// TIA Portal V20 export
FUNCTION_BLOCK "FB_Send_Water_Fountain_To_Rework"   // FB7, LAD
{ S7_Optimized_Access := 'TRUE' }
// stored: AutoNumber false, MemoryReserve 100, SetENOAutomatically false
   VAR_INPUT
      Emergency_Stop_Release : Bool;
      Start : Bool;
      Water_Fountain_Fail_Test : Bool;
      Trigger_Read_Serial_Number_Exit_Functional_Test : Bool;
      Sensor_Water_Fountain_Exit_Functional_Test_Spinner_Conveyor_Belt : Bool;
      Sensor_Spinner_Exit_Functional_Test_Position_Withdrawn : Bool;
      Sensor_Spinner_Exit_Functional_Test_Position_Advanced : Bool;
      Sensor_Water_Fountain_Exit_Functional_Test_After_Spinner_Conveyor_Belt : Bool;
      Sensor_Water_Fountain_Geting_Entrace_Rework_Conveyor_Belt_Start : Bool;
   END_VAR
   VAR_OUTPUT
      Turn_On_Conveyor_Belt_Motor_Spinner_Get_Exit_Functional_Test : Bool;
      Valve_Advance_Spinner_Get_Exit_Functional_Test : Bool;
      Pause_Conveyor_Belt_And_Carousel_Functional_Test : Bool;
   END_VAR
   VAR
      Aux_Trig_0 : Bool;
      Aux_Trig_1 : Bool;
      Aux_Trig_2 : Bool;
      Aux_Trig_3 : Bool;
      Aux_Trig_4 : Bool;
      Aux_Trig_5 : Bool;
      Aux_Trig_6 : Bool;
      Aux_Trig_7 : Bool;
      Wait_Clean_Spinner : Bool;
      Wait_Get_In_Spinner : Bool;
      "Counter" : USInt;
      Timer_Delay_Turn_On_Motor_Spinner_Conveyor_Belt { S7_SetPoint := 'True'} : TON_TIME;
   END_VAR
   VAR RETAIN
      Counter_Water_Fountain_Exiting_Functional_Test { S7_SetPoint := 'True'} : CTUD_USINT;
   END_VAR
   VAR_TEMP   // added for the SCL form of the ladder/FBD networks
      _w1 : Bool;
      _w2 : Bool;
   END_VAR
BEGIN

REGION Network 1
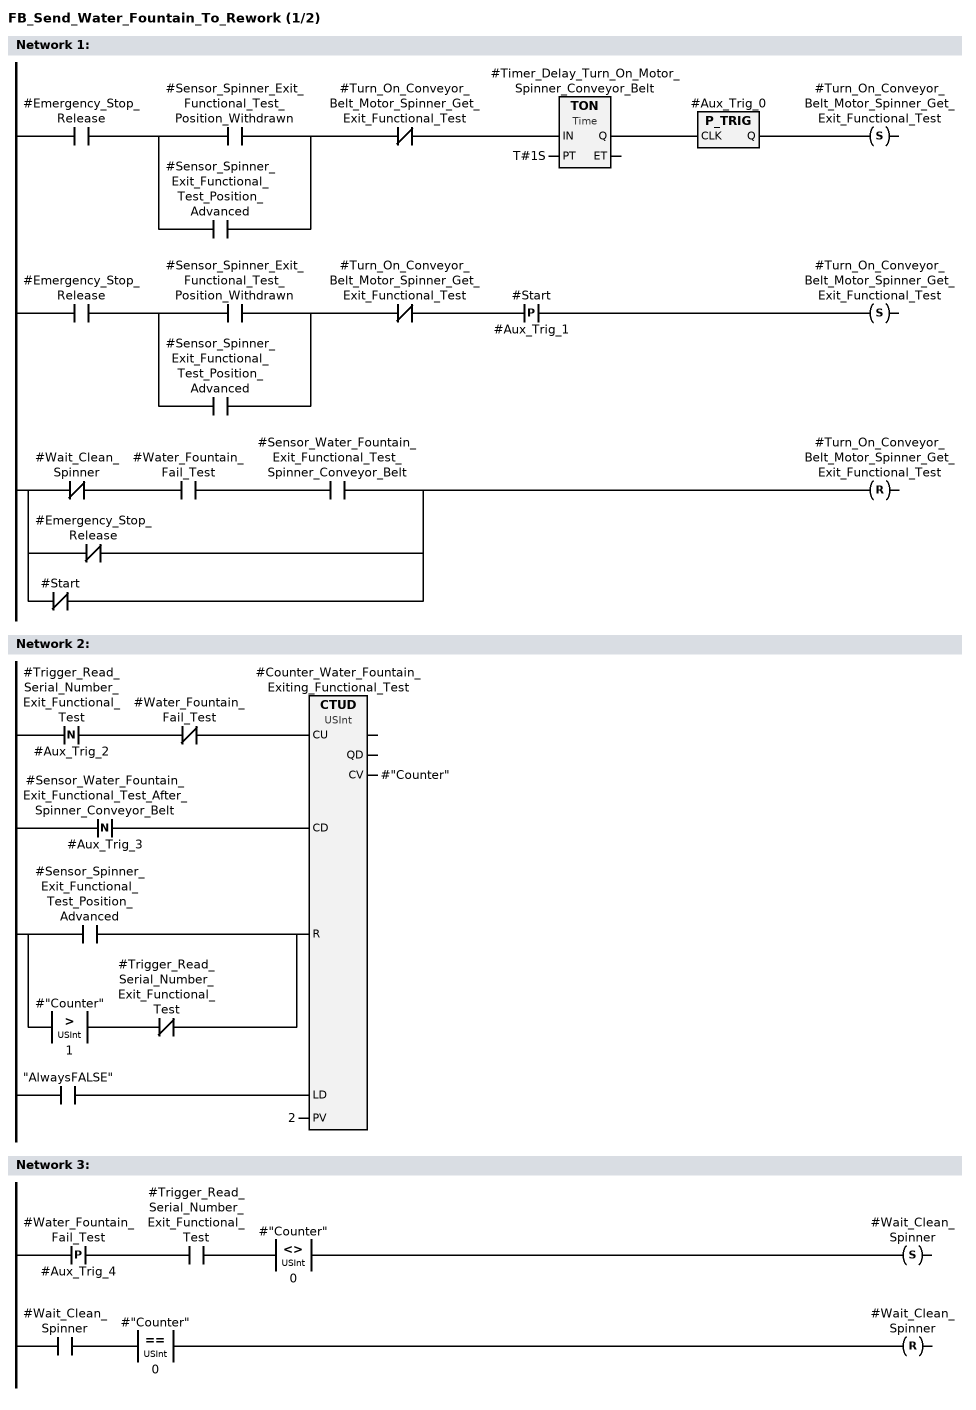
   RUNG wire#powerrail
      Contact( #Emergency_Stop_Release )
      wire#w1
      Contact( #Sensor_Spinner_Exit_Functional_Test_Position_Withdrawn )
      wire#w2
      I_Contact( #Turn_On_Conveyor_Belt_Motor_Spinner_Get_Exit_Functional_Test )
      { S7_Templates := "time_type := Time" } #Timer_Delay_Turn_On_Motor_Spinner_Conveyor_Belt.TON(pt := T#1S, et =>)
      P_Trig( #Aux_Trig_0 )
      S_Coil( #Turn_On_Conveyor_Belt_Motor_Spinner_Get_Exit_Functional_Test )
   END_RUNG
   RUNG wire#w1
      Contact( #Sensor_Spinner_Exit_Functional_Test_Position_Advanced )
   END_RUNG wire#w2
   RUNG wire#powerrail
      Contact( #Emergency_Stop_Release )
      wire#w3
      Contact( #Sensor_Spinner_Exit_Functional_Test_Position_Withdrawn )
      wire#w4
      I_Contact( #Turn_On_Conveyor_Belt_Motor_Spinner_Get_Exit_Functional_Test )
      P_Contact(operand := #Start, bit := #Aux_Trig_1)
      S_Coil( #Turn_On_Conveyor_Belt_Motor_Spinner_Get_Exit_Functional_Test )
   END_RUNG
   RUNG wire#w3
      Contact( #Sensor_Spinner_Exit_Functional_Test_Position_Advanced )
   END_RUNG wire#w4
   RUNG wire#powerrail
      I_Contact( #Wait_Clean_Spinner )
      Contact( #Water_Fountain_Fail_Test )
      Contact( #Sensor_Water_Fountain_Exit_Functional_Test_Spinner_Conveyor_Belt )
      wire#w5
      R_Coil( #Turn_On_Conveyor_Belt_Motor_Spinner_Get_Exit_Functional_Test )
   END_RUNG
   RUNG wire#powerrail
      I_Contact( #Emergency_Stop_Release )
   END_RUNG wire#w5
   RUNG wire#powerrail
      I_Contact( #Start )
   END_RUNG wire#w5
   // the same network as SCL:
   #Timer_Delay_Turn_On_Motor_Spinner_Conveyor_Belt(IN := #Emergency_Stop_Release AND (#Sensor_Spinner_Exit_Functional_Test_Position_Withdrawn OR #Sensor_Spinner_Exit_Functional_Test_Position_Advanced) AND NOT #Turn_On_Conveyor_Belt_Motor_Spinner_Get_Exit_Functional_Test,   // TON
                           PT := T#1S);
   #_w1 := #Timer_Delay_Turn_On_Motor_Spinner_Conveyor_Belt.Q AND NOT #Aux_Trig_0;   // rising edge
   #Aux_Trig_0 := #Timer_Delay_Turn_On_Motor_Spinner_Conveyor_Belt.Q;
   IF #_w1 THEN #Turn_On_Conveyor_Belt_Motor_Spinner_Get_Exit_Functional_Test := TRUE; END_IF;
   #_w2 := #Emergency_Stop_Release AND (#Sensor_Spinner_Exit_Functional_Test_Position_Withdrawn OR #Sensor_Spinner_Exit_Functional_Test_Position_Advanced) AND NOT #Turn_On_Conveyor_Belt_Motor_Spinner_Get_Exit_Functional_Test AND #Start AND NOT #Aux_Trig_1;   // rising edge of #Start
   #Aux_Trig_1 := #Start;
   IF #_w2 THEN #Turn_On_Conveyor_Belt_Motor_Spinner_Get_Exit_Functional_Test := TRUE; END_IF;
   IF (NOT #Wait_Clean_Spinner AND #Water_Fountain_Fail_Test AND #Sensor_Water_Fountain_Exit_Functional_Test_Spinner_Conveyor_Belt) OR NOT #Emergency_Stop_Release OR NOT #Start THEN
       #Turn_On_Conveyor_Belt_Motor_Spinner_Get_Exit_Functional_Test := FALSE;
   END_IF;
END_REGION

REGION Network 2
   RUNG wire#powerrail
      N_Contact(operand := #Trigger_Read_Serial_Number_Exit_Functional_Test, bit := #Aux_Trig_2)
      I_Contact( #Water_Fountain_Fail_Test )
      { S7_Templates := "value_type := USInt" } #Counter_Water_Fountain_Exiting_Functional_Test.CTUD(cd := wire#w1, r := wire#w2, ld := wire#w3, pv := 2, qd =>, cv => #"Counter")
   END_RUNG
   RUNG wire#powerrail
      N_Contact(operand := #Sensor_Water_Fountain_Exit_Functional_Test_After_Spinner_Conveyor_Belt, bit := #Aux_Trig_3)
   END_RUNG wire#w1
   RUNG wire#powerrail
      Contact( #Sensor_Spinner_Exit_Functional_Test_Position_Advanced )
   END_RUNG wire#w2
   RUNG wire#powerrail
      { S7_Templates := "SrcType := USInt" } GT_Contact(in1 := #"Counter", in2 := 1)
      I_Contact( #Trigger_Read_Serial_Number_Exit_Functional_Test )
   END_RUNG wire#w2
   RUNG wire#powerrail
      Contact( "AlwaysFALSE" )
   END_RUNG wire#w3
   // the same network as SCL:
   #_w1 := NOT #Trigger_Read_Serial_Number_Exit_Functional_Test AND #Aux_Trig_2;   // falling edge of #Trigger_Read_Serial_Number_Exit_Functional_Test
   #Aux_Trig_2 := #Trigger_Read_Serial_Number_Exit_Functional_Test;
   #_w2 := NOT #Sensor_Water_Fountain_Exit_Functional_Test_After_Spinner_Conveyor_Belt AND #Aux_Trig_3;   // falling edge of #Sensor_Water_Fountain_Exit_Functional_Test_After_Spinner_Conveyor_Belt
   #Aux_Trig_3 := #Sensor_Water_Fountain_Exit_Functional_Test_After_Spinner_Conveyor_Belt;
   #Counter_Water_Fountain_Exiting_Functional_Test(CU := #_w1 AND NOT #Water_Fountain_Fail_Test,   // CTUD
                           CD := #_w2,
                           R := #Sensor_Spinner_Exit_Functional_Test_Position_Advanced OR ((#"Counter" > 1) AND NOT #Trigger_Read_Serial_Number_Exit_Functional_Test),
                           LD := "AlwaysFALSE",
                           PV := 2,
                           CV => #"Counter");
END_REGION

REGION Network 3
   RUNG wire#powerrail
      P_Contact(operand := #Water_Fountain_Fail_Test, bit := #Aux_Trig_4)
      Contact( #Trigger_Read_Serial_Number_Exit_Functional_Test )
      { S7_Templates := "SrcType := USInt" } NE_Contact(in1 := #"Counter", in2 := 0)
      S_Coil( #Wait_Clean_Spinner )
   END_RUNG
   RUNG wire#powerrail
      Contact( #Wait_Clean_Spinner )
      { S7_Templates := "SrcType := USInt" } EQ_Contact(in1 := #"Counter", in2 := 0)
      R_Coil( #Wait_Clean_Spinner )
   END_RUNG
   // the same network as SCL:
   #_w1 := #Water_Fountain_Fail_Test AND NOT #Aux_Trig_4;   // rising edge of #Water_Fountain_Fail_Test
   #Aux_Trig_4 := #Water_Fountain_Fail_Test;
   IF #_w1 AND #Trigger_Read_Serial_Number_Exit_Functional_Test AND (#"Counter" <> 0) THEN
       #Wait_Clean_Spinner := TRUE;
   END_IF;
   IF #Wait_Clean_Spinner AND (#"Counter" = 0) THEN #Wait_Clean_Spinner := FALSE; END_IF;
END_REGION

REGION Network 4
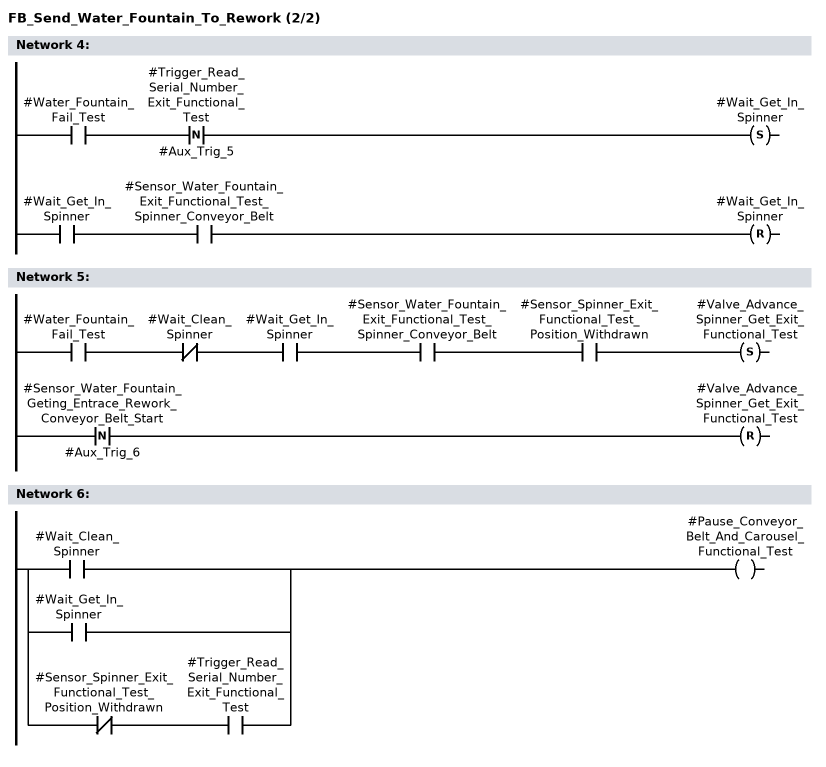
   RUNG wire#powerrail
      Contact( #Water_Fountain_Fail_Test )
      N_Contact(operand := #Trigger_Read_Serial_Number_Exit_Functional_Test, bit := #Aux_Trig_5)
      S_Coil( #Wait_Get_In_Spinner )
   END_RUNG
   RUNG wire#powerrail
      Contact( #Wait_Get_In_Spinner )
      Contact( #Sensor_Water_Fountain_Exit_Functional_Test_Spinner_Conveyor_Belt )
      R_Coil( #Wait_Get_In_Spinner )
   END_RUNG
   // the same network as SCL:
   #_w1 := #Water_Fountain_Fail_Test AND NOT #Trigger_Read_Serial_Number_Exit_Functional_Test AND #Aux_Trig_5;   // falling edge of #Trigger_Read_Serial_Number_Exit_Functional_Test
   #Aux_Trig_5 := #Trigger_Read_Serial_Number_Exit_Functional_Test;
   IF #_w1 THEN #Wait_Get_In_Spinner := TRUE; END_IF;
   IF #Wait_Get_In_Spinner AND #Sensor_Water_Fountain_Exit_Functional_Test_Spinner_Conveyor_Belt THEN
       #Wait_Get_In_Spinner := FALSE;
   END_IF;
END_REGION

REGION Network 5
   RUNG wire#powerrail
      Contact( #Water_Fountain_Fail_Test )
      I_Contact( #Wait_Clean_Spinner )
      Contact( #Wait_Get_In_Spinner )
      Contact( #Sensor_Water_Fountain_Exit_Functional_Test_Spinner_Conveyor_Belt )
      Contact( #Sensor_Spinner_Exit_Functional_Test_Position_Withdrawn )
      S_Coil( #Valve_Advance_Spinner_Get_Exit_Functional_Test )
   END_RUNG
   RUNG wire#powerrail
      N_Contact(operand := #Sensor_Water_Fountain_Geting_Entrace_Rework_Conveyor_Belt_Start, bit := #Aux_Trig_6)
      R_Coil( #Valve_Advance_Spinner_Get_Exit_Functional_Test )
   END_RUNG
   // the same network as SCL:
   IF #Water_Fountain_Fail_Test AND NOT #Wait_Clean_Spinner AND #Wait_Get_In_Spinner AND #Sensor_Water_Fountain_Exit_Functional_Test_Spinner_Conveyor_Belt AND #Sensor_Spinner_Exit_Functional_Test_Position_Withdrawn THEN
       #Valve_Advance_Spinner_Get_Exit_Functional_Test := TRUE;
   END_IF;
   #_w1 := NOT #Sensor_Water_Fountain_Geting_Entrace_Rework_Conveyor_Belt_Start AND #Aux_Trig_6;   // falling edge of #Sensor_Water_Fountain_Geting_Entrace_Rework_Conveyor_Belt_Start
   #Aux_Trig_6 := #Sensor_Water_Fountain_Geting_Entrace_Rework_Conveyor_Belt_Start;
   IF #_w1 THEN #Valve_Advance_Spinner_Get_Exit_Functional_Test := FALSE; END_IF;
END_REGION

REGION Network 6
   RUNG wire#powerrail
      Contact( #Wait_Clean_Spinner )
      wire#w1
      Coil( #Pause_Conveyor_Belt_And_Carousel_Functional_Test )
   END_RUNG
   RUNG wire#powerrail
      Contact( #Wait_Get_In_Spinner )
   END_RUNG wire#w1
   RUNG wire#powerrail
      I_Contact( #Sensor_Spinner_Exit_Functional_Test_Position_Withdrawn )
      Contact( #Trigger_Read_Serial_Number_Exit_Functional_Test )
   END_RUNG wire#w1
   // the same network as SCL:
   #Pause_Conveyor_Belt_And_Carousel_Functional_Test := #Wait_Clean_Spinner OR #Wait_Get_In_Spinner OR (NOT #Sensor_Spinner_Exit_Functional_Test_Position_Withdrawn AND #Trigger_Read_Serial_Number_Exit_Functional_Test);
END_REGION
END_FUNCTION_BLOCK
